// SIMATIC S7-200 project (STEP 7-Micro/WIN), CPU 224XP REL 02.01

SYMBOL_TABLE USUARIO1
PULSADOR_SUMA    I0.0     // ASCENDENTE
PULSADOR_RESTA   I0.1     // DESCENDENTE
RESET            I0.2     // RESET(REPRESENTA 0)
DISPLAY_1        MB10
DISPLAY_2        MB11
CONTADOR_1       MW2
CONTADOR_2       MW4
SEGMENTO_0_D1    Q0.0
SEGMENTO_1_D1    Q0.1
SEGMENTO_2_D1    Q0.2
SEGMENTO_3_D1    Q0.3
SEGMENTO_4_D1    Q0.4
SEGMENTO_5_D1    Q0.5
SEGMENTO_6_D1    Q0.6
SEGMENTO_0_D2    Q1.0
SEGMENTO_1_D2    Q1.1
SEGMENTO_2_D2    Q1.2
SEGMENTO_3_D2    Q1.3
SEGMENTO_4_D2    Q1.4
SEGMENTO_5_D2    Q1.5
SEGMENTO_6_D2    Q1.6
END_SYMBOL_TABLE

SYMBOL_TABLE Símbolos S7-200
Siempre_ON       SM0.0    // Siempre ON
Primer_ciclo_ON  SM0.1    // ON sólo en el primer ciclo
END_SYMBOL_TABLE

ORGANIZATION_BLOCK PRINCIPAL:OB1
TITLE=COMENTARIOS DEL PROGRAMA
BEGIN
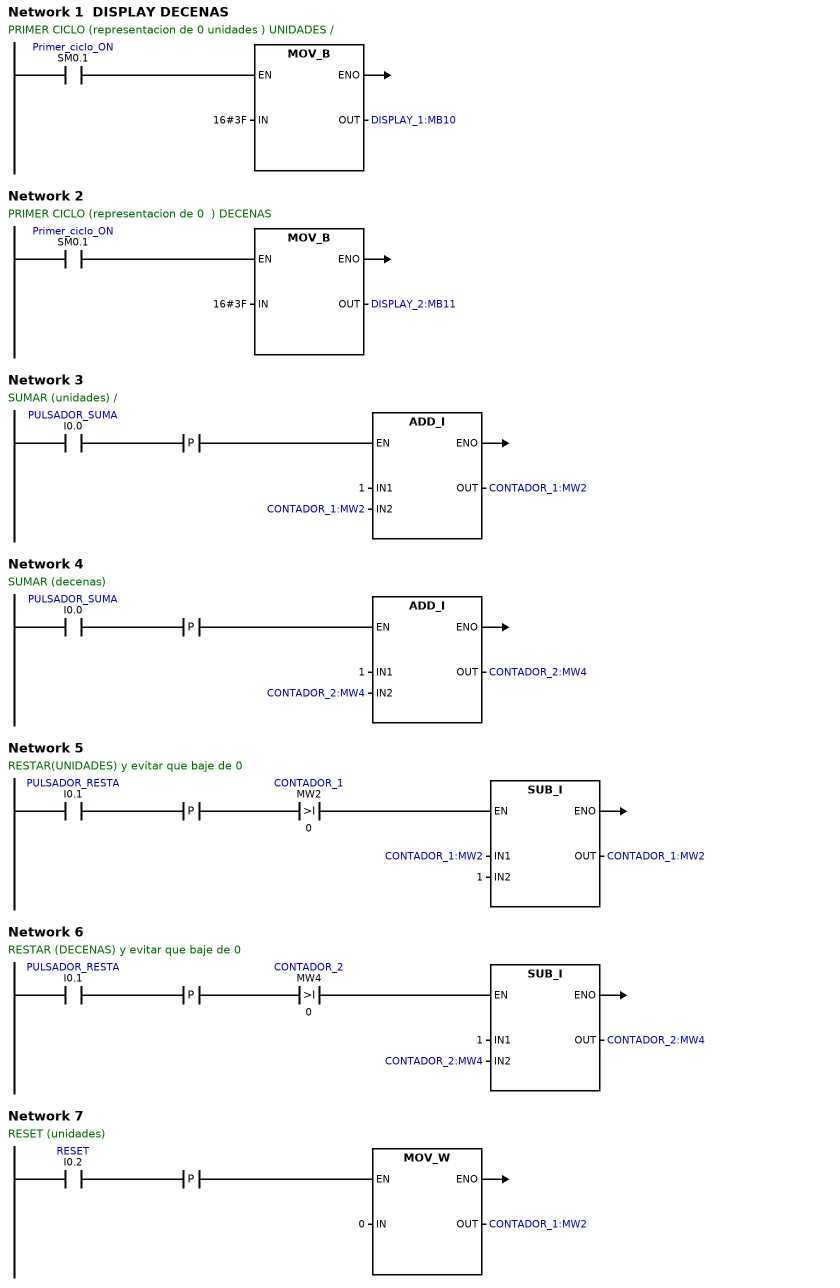
Network 1 // DISPLAY DECENAS
// PRIMER CICLO (representacion de 0 unidades ) UNIDADES
// 
LD     Primer_ciclo_ON:SM0.1
MOVB   16#3F, DISPLAY_1:MB10
Network 2
// PRIMER CICLO (representacion de 0  ) DECENAS
LD     Primer_ciclo_ON:SM0.1
MOVB   16#3F, DISPLAY_2:MB11
Network 3
// SUMAR (unidades)
// 
// (network saved uncompiled; LAD cells follow)
// row 0: c0 -| |- PULSADOR_SUMA:I0.0  c1 -|P|-  c2 --  c3 [ADD_I EN:=power@row0, IN1:=1, IN2:=CONTADOR_1:MW2, ENO=>power, OUT=>CONTADOR_1:MW2]  c4 ->
// row 1: c3 [box]
Network 4
// SUMAR (decenas)
// (network saved uncompiled; LAD cells follow)
// row 0: c0 -| |- PULSADOR_SUMA:I0.0  c1 -|P|-  c2 --  c3 [ADD_I EN:=power@row0, IN1:=1, IN2:=CONTADOR_2:MW4, ENO=>power, OUT=>CONTADOR_2:MW4]  c4 ->
// row 1: c3 [box]
Network 5
// RESTAR(UNIDADES) y evitar que baje de 0
// (network saved uncompiled; LAD cells follow)
// row 0: c0 -| |- PULSADOR_RESTA:I0.1  c1 -|P|-  c2 -|>I|- CONTADOR_1:MW2, 0  c3 --  c4 [SUB_I EN:=power@row0, IN1:=CONTADOR_1:MW2, IN2:=1, ENO=>power, OUT=>CONTADOR_1:MW2]  c5 ->
// row 1: c4 [box]
Network 6
// RESTAR (DECENAS) y evitar que baje de 0
// (network saved uncompiled; LAD cells follow)
// row 0: c0 -| |- PULSADOR_RESTA:I0.1  c1 -|P|-  c2 -|>I|- CONTADOR_2:MW4, 0  c3 --  c4 [SUB_I EN:=power@row0, IN1:=1, IN2:=CONTADOR_2:MW4, ENO=>power, OUT=>CONTADOR_2:MW4]  c5 ->
// row 1: c4 [box]
Network 7
// RESET (unidades)
// (network saved uncompiled; LAD cells follow)
// row 0: c0 -| |- RESET:I0.2  c1 -|P|-  c2 --  c3 [MOV_W EN:=power@row0, IN:=0, ENO=>power, OUT=>CONTADOR_1:MW2]  c4 ->
// row 1: c3 [box]
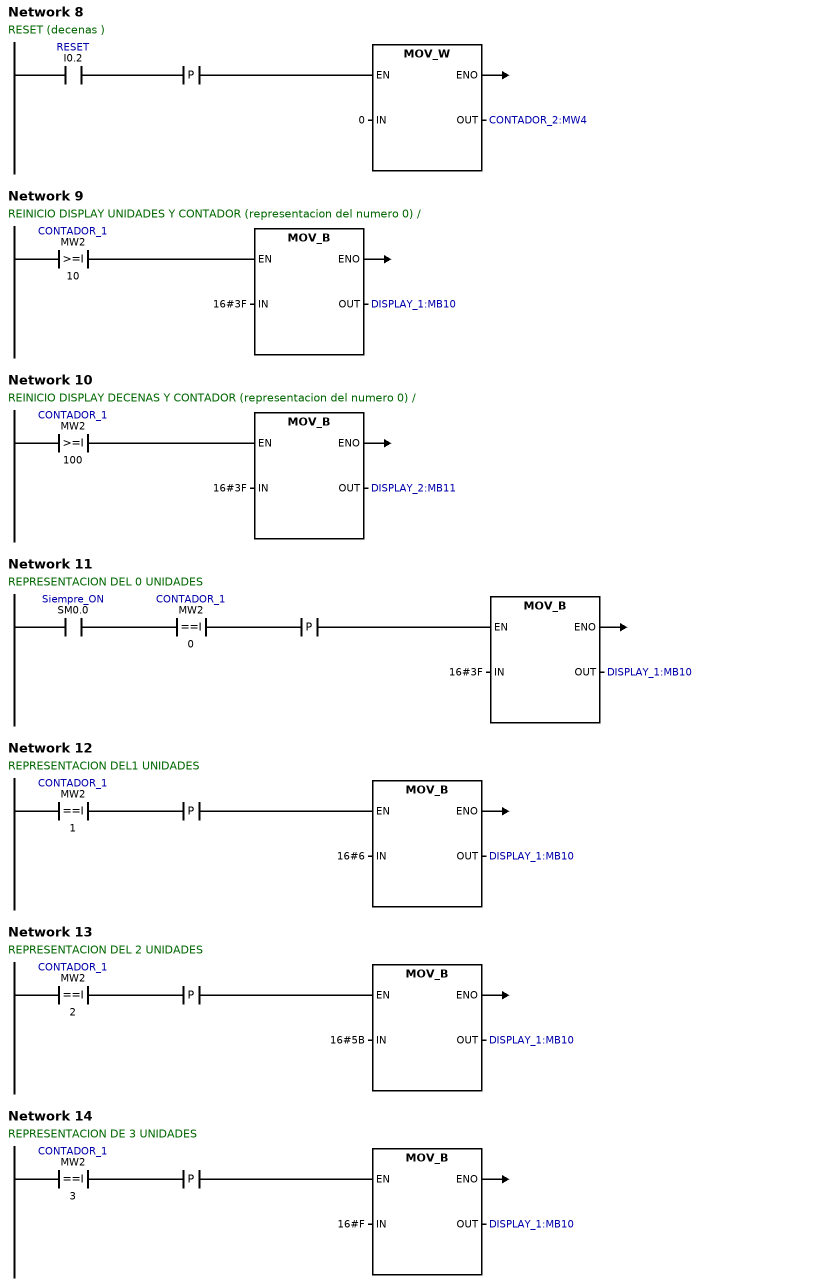
Network 8
// RESET (decenas )
// (network saved uncompiled; LAD cells follow)
// row 0: c0 -| |- RESET:I0.2  c1 -|P|-  c2 --  c3 [MOV_W EN:=power@row0, IN:=0, ENO=>power, OUT=>CONTADOR_2:MW4]  c4 ->
// row 1: c3 [box]
Network 9
// REINICIO DISPLAY UNIDADES Y CONTADOR (representacion del numero 0)
// 
// (network saved uncompiled; LAD cells follow)
// row 0: c0 -|>=I|- CONTADOR_1:MW2, 10  c1 --  c2 [MOV_B EN:=power@row0, IN:=16#3F, ENO=>power, OUT=>DISPLAY_1:MB10]  c3 ->
// row 1: c2 [box]
Network 10
// REINICIO DISPLAY DECENAS Y CONTADOR (representacion del numero 0)
// 
// (network saved uncompiled; LAD cells follow)
// row 0: c0 -|>=I|- CONTADOR_1:MW2, 100  c1 --  c2 [MOV_B EN:=power@row0, IN:=16#3F, ENO=>power, OUT=>DISPLAY_2:MB11]  c3 ->
// row 1: c2 [box]
Network 11
// REPRESENTACION DEL 0 UNIDADES
// (network saved uncompiled; LAD cells follow)
// row 0: c0 -| |- Siempre_ON:SM0.0  c1 -|==I|- CONTADOR_1:MW2, 0  c2 -|P|-  c3 --  c4 [MOV_B EN:=power@row0, IN:=16#3F, ENO=>power, OUT=>DISPLAY_1:MB10]  c5 ->
// row 1: c4 [box]
Network 12
// REPRESENTACION DEL1 UNIDADES
// (network saved uncompiled; LAD cells follow)
// row 0: c0 -|==I|- CONTADOR_1:MW2, 1  c1 -|P|-  c2 --  c3 [MOV_B EN:=power@row0, IN:=16#6, ENO=>power, OUT=>DISPLAY_1:MB10]  c4 ->
// row 1: c3 [box]
Network 13
// REPRESENTACION DEL 2 UNIDADES
// (network saved uncompiled; LAD cells follow)
// row 0: c0 -|==I|- CONTADOR_1:MW2, 2  c1 -|P|-  c2 --  c3 [MOV_B EN:=power@row0, IN:=16#5B, ENO=>power, OUT=>DISPLAY_1:MB10]  c4 ->
// row 1: c3 [box]
Network 14
// REPRESENTACION DE 3 UNIDADES
// (network saved uncompiled; LAD cells follow)
// row 0: c0 -|==I|- CONTADOR_1:MW2, 3  c1 -|P|-  c2 --  c3 [MOV_B EN:=power@row0, IN:=16#F, ENO=>power, OUT=>DISPLAY_1:MB10]  c4 ->
// row 1: c3 [box]
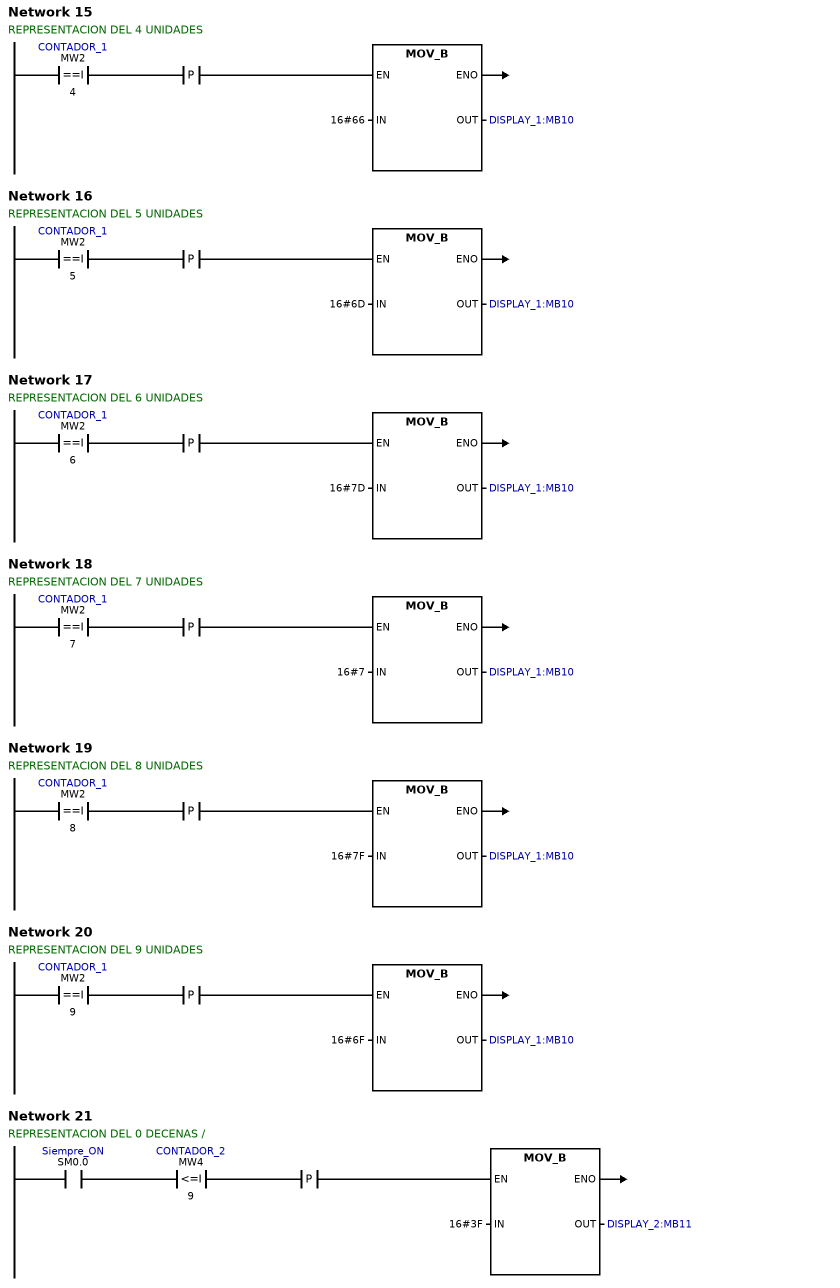
Network 15
// REPRESENTACION DEL 4 UNIDADES
// (network saved uncompiled; LAD cells follow)
// row 0: c0 -|==I|- CONTADOR_1:MW2, 4  c1 -|P|-  c2 --  c3 [MOV_B EN:=power@row0, IN:=16#66, ENO=>power, OUT=>DISPLAY_1:MB10]  c4 ->
// row 1: c3 [box]
Network 16
// REPRESENTACION DEL 5 UNIDADES
// (network saved uncompiled; LAD cells follow)
// row 0: c0 -|==I|- CONTADOR_1:MW2, 5  c1 -|P|-  c2 --  c3 [MOV_B EN:=power@row0, IN:=16#6D, ENO=>power, OUT=>DISPLAY_1:MB10]  c4 ->
// row 1: c3 [box]
Network 17
// REPRESENTACION DEL 6 UNIDADES
// (network saved uncompiled; LAD cells follow)
// row 0: c0 -|==I|- CONTADOR_1:MW2, 6  c1 -|P|-  c2 --  c3 [MOV_B EN:=power@row0, IN:=16#7D, ENO=>power, OUT=>DISPLAY_1:MB10]  c4 ->
// row 1: c3 [box]
Network 18
// REPRESENTACION DEL 7 UNIDADES
// (network saved uncompiled; LAD cells follow)
// row 0: c0 -|==I|- CONTADOR_1:MW2, 7  c1 -|P|-  c2 --  c3 [MOV_B EN:=power@row0, IN:=16#7, ENO=>power, OUT=>DISPLAY_1:MB10]  c4 ->
// row 1: c3 [box]
Network 19
// REPRESENTACION DEL 8 UNIDADES
// (network saved uncompiled; LAD cells follow)
// row 0: c0 -|==I|- CONTADOR_1:MW2, 8  c1 -|P|-  c2 --  c3 [MOV_B EN:=power@row0, IN:=16#7F, ENO=>power, OUT=>DISPLAY_1:MB10]  c4 ->
// row 1: c3 [box]
Network 20
// REPRESENTACION DEL 9 UNIDADES
// (network saved uncompiled; LAD cells follow)
// row 0: c0 -|==I|- CONTADOR_1:MW2, 9  c1 -|P|-  c2 --  c3 [MOV_B EN:=power@row0, IN:=16#6F, ENO=>power, OUT=>DISPLAY_1:MB10]  c4 ->
// row 1: c3 [box]
Network 21
// REPRESENTACION DEL 0 DECENAS
// 
// (network saved uncompiled; LAD cells follow)
// row 0: c0 -| |- Siempre_ON:SM0.0  c1 -|<=I|- CONTADOR_2:MW4, 9  c2 -|P|-  c3 --  c4 [MOV_B EN:=power@row0, IN:=16#3F, ENO=>power, OUT=>DISPLAY_2:MB11]  c5 ->
// row 1: c4 [box]
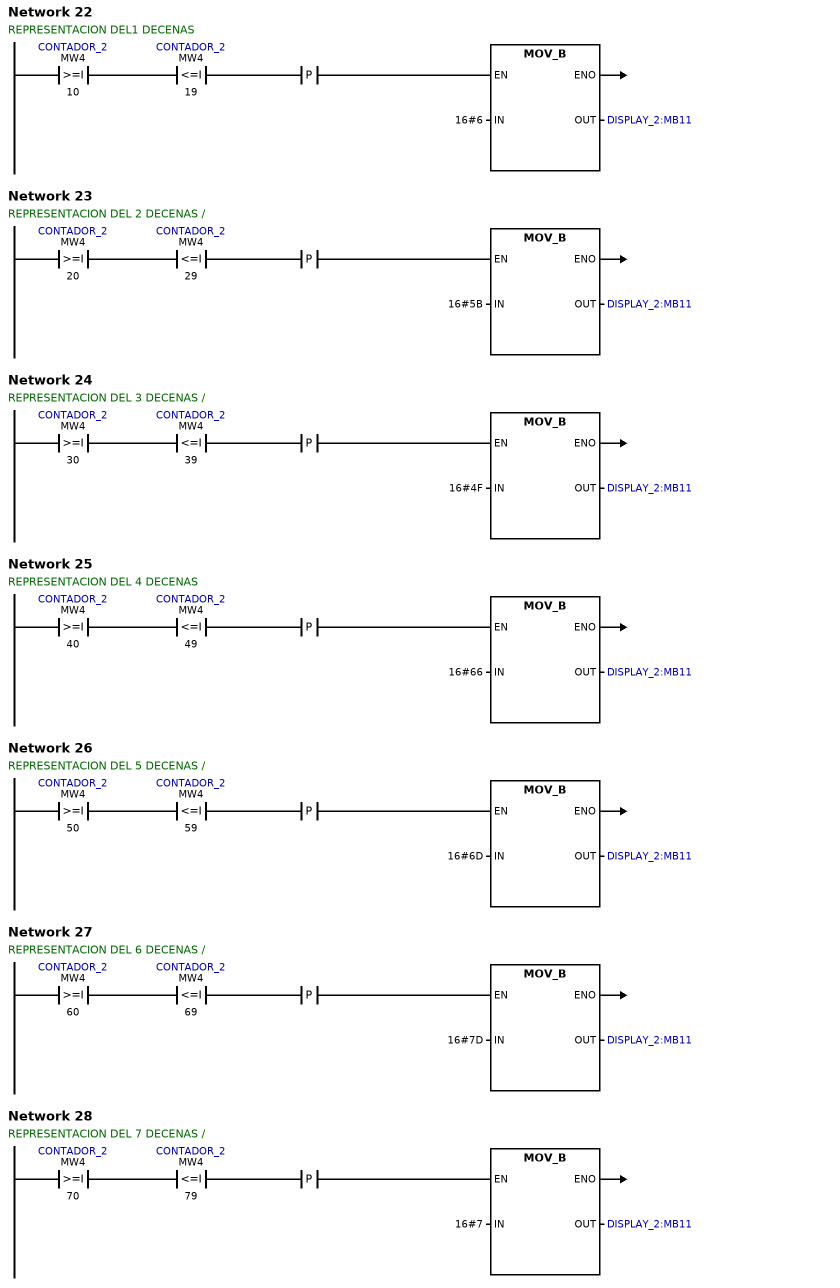
Network 22
// REPRESENTACION DEL1 DECENAS
// (network saved uncompiled; LAD cells follow)
// row 0: c0 -|>=I|- CONTADOR_2:MW4, 10  c1 -|<=I|- CONTADOR_2:MW4, 19  c2 -|P|-  c3 --  c4 [MOV_B EN:=power@row0, IN:=16#6, ENO=>power, OUT=>DISPLAY_2:MB11]  c5 ->
// row 1: c4 [box]
Network 23
// REPRESENTACION DEL 2 DECENAS
// 
// (network saved uncompiled; LAD cells follow)
// row 0: c0 -|>=I|- CONTADOR_2:MW4, 20  c1 -|<=I|- CONTADOR_2:MW4, 29  c2 -|P|-  c3 --  c4 [MOV_B EN:=power@row0, IN:=16#5B, ENO=>power, OUT=>DISPLAY_2:MB11]  c5 ->
// row 1: c4 [box]
Network 24
// REPRESENTACION DEL 3 DECENAS
// 
// (network saved uncompiled; LAD cells follow)
// row 0: c0 -|>=I|- CONTADOR_2:MW4, 30  c1 -|<=I|- CONTADOR_2:MW4, 39  c2 -|P|-  c3 --  c4 [MOV_B EN:=power@row0, IN:=16#4F, ENO=>power, OUT=>DISPLAY_2:MB11]  c5 ->
// row 1: c4 [box]
Network 25
// REPRESENTACION DEL 4 DECENAS
// (network saved uncompiled; LAD cells follow)
// row 0: c0 -|>=I|- CONTADOR_2:MW4, 40  c1 -|<=I|- CONTADOR_2:MW4, 49  c2 -|P|-  c3 --  c4 [MOV_B EN:=power@row0, IN:=16#66, ENO=>power, OUT=>DISPLAY_2:MB11]  c5 ->
// row 1: c4 [box]
Network 26
// REPRESENTACION DEL 5 DECENAS
// 
// (network saved uncompiled; LAD cells follow)
// row 0: c0 -|>=I|- CONTADOR_2:MW4, 50  c1 -|<=I|- CONTADOR_2:MW4, 59  c2 -|P|-  c3 --  c4 [MOV_B EN:=power@row0, IN:=16#6D, ENO=>power, OUT=>DISPLAY_2:MB11]  c5 ->
// row 1: c4 [box]
Network 27
// REPRESENTACION DEL 6 DECENAS
// 
// (network saved uncompiled; LAD cells follow)
// row 0: c0 -|>=I|- CONTADOR_2:MW4, 60  c1 -|<=I|- CONTADOR_2:MW4, 69  c2 -|P|-  c3 --  c4 [MOV_B EN:=power@row0, IN:=16#7D, ENO=>power, OUT=>DISPLAY_2:MB11]  c5 ->
// row 1: c4 [box]
Network 28
// REPRESENTACION DEL 7 DECENAS
// 
// (network saved uncompiled; LAD cells follow)
// row 0: c0 -|>=I|- CONTADOR_2:MW4, 70  c1 -|<=I|- CONTADOR_2:MW4, 79  c2 -|P|-  c3 --  c4 [MOV_B EN:=power@row0, IN:=16#7, ENO=>power, OUT=>DISPLAY_2:MB11]  c5 ->
// row 1: c4 [box]
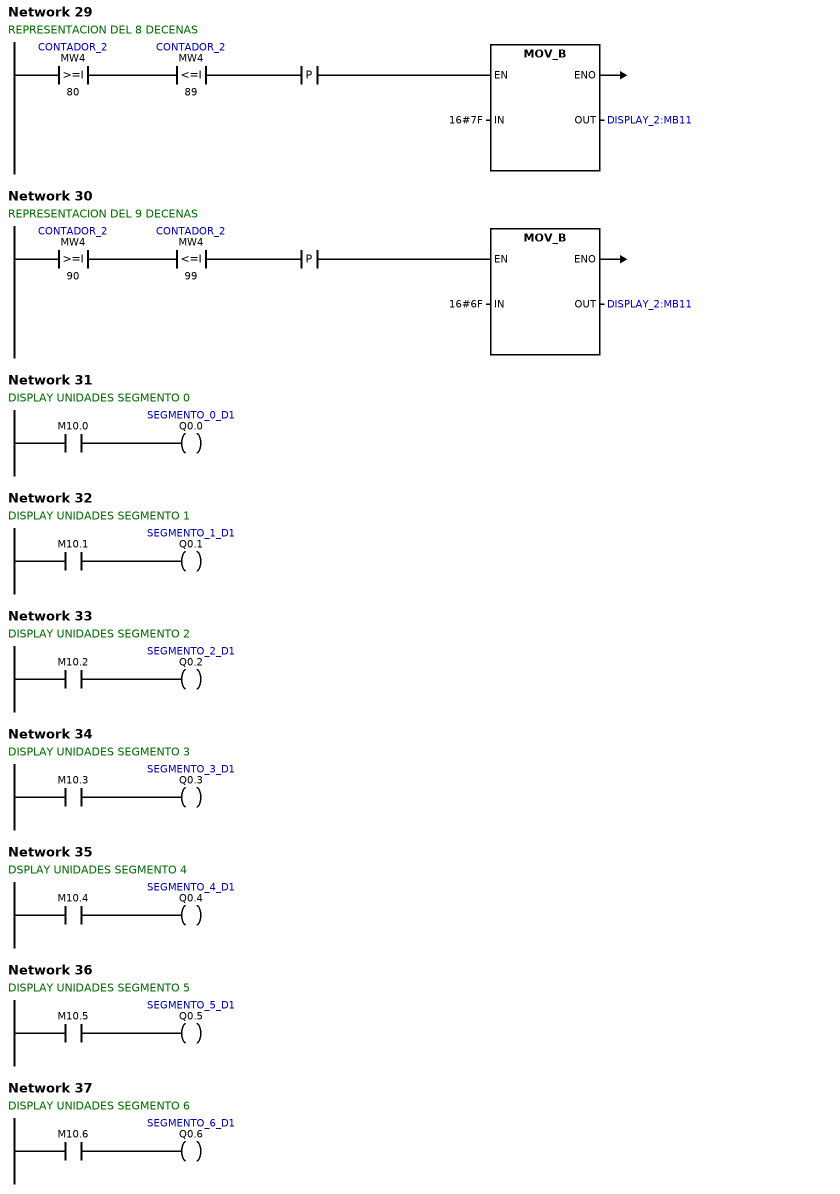
Network 29
// REPRESENTACION DEL 8 DECENAS
// (network saved uncompiled; LAD cells follow)
// row 0: c0 -|>=I|- CONTADOR_2:MW4, 80  c1 -|<=I|- CONTADOR_2:MW4, 89  c2 -|P|-  c3 --  c4 [MOV_B EN:=power@row0, IN:=16#7F, ENO=>power, OUT=>DISPLAY_2:MB11]  c5 ->
// row 1: c4 [box]
Network 30
// REPRESENTACION DEL 9 DECENAS
// (network saved uncompiled; LAD cells follow)
// row 0: c0 -|>=I|- CONTADOR_2:MW4, 90  c1 -|<=I|- CONTADOR_2:MW4, 99  c2 -|P|-  c3 --  c4 [MOV_B EN:=power@row0, IN:=16#6F, ENO=>power, OUT=>DISPLAY_2:MB11]  c5 ->
// row 1: c4 [box]
Network 31
// DISPLAY UNIDADES SEGMENTO 0
LD     M10.0
=      SEGMENTO_0_D1:Q0.0
Network 32
// DISPLAY UNIDADES SEGMENTO 1
LD     M10.1
=      SEGMENTO_1_D1:Q0.1
Network 33
// DISPLAY UNIDADES SEGMENTO 2
LD     M10.2
=      SEGMENTO_2_D1:Q0.2
Network 34
// DISPLAY UNIDADES SEGMENTO 3
LD     M10.3
=      SEGMENTO_3_D1:Q0.3
Network 35
// DSPLAY UNIDADES SEGMENTO 4
LD     M10.4
=      SEGMENTO_4_D1:Q0.4
Network 36
// DISPLAY UNIDADES SEGMENTO 5
LD     M10.5
=      SEGMENTO_5_D1:Q0.5
Network 37
// DISPLAY UNIDADES SEGMENTO 6
LD     M10.6
=      SEGMENTO_6_D1:Q0.6
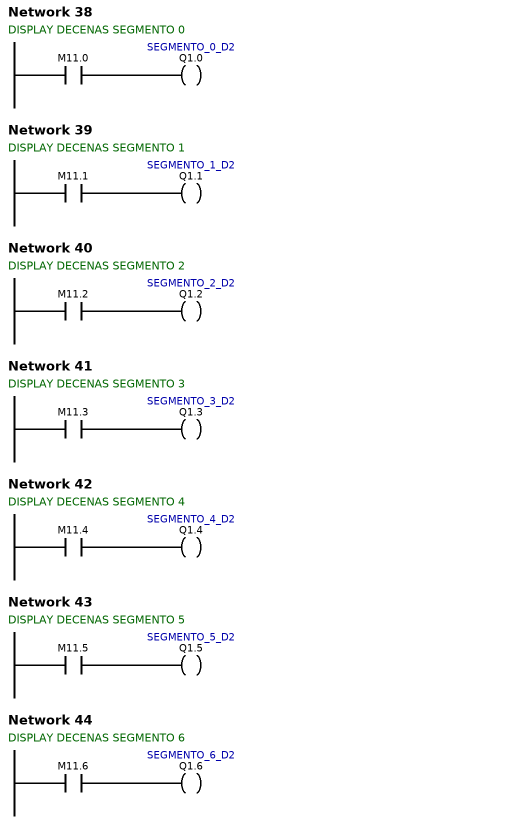
Network 38
// DISPLAY DECENAS SEGMENTO 0
LD     M11.0
=      SEGMENTO_0_D2:Q1.0
Network 39
// DISPLAY DECENAS SEGMENTO 1
LD     M11.1
=      SEGMENTO_1_D2:Q1.1
Network 40
// DISPLAY DECENAS SEGMENTO 2
LD     M11.2
=      SEGMENTO_2_D2:Q1.2
Network 41
// DISPLAY DECENAS SEGMENTO 3
LD     M11.3
=      SEGMENTO_3_D2:Q1.3
Network 42
// DISPLAY DECENAS SEGMENTO 4
LD     M11.4
=      SEGMENTO_4_D2:Q1.4
Network 43
// DISPLAY DECENAS SEGMENTO 5
LD     M11.5
=      SEGMENTO_5_D2:Q1.5
Network 44
// DISPLAY DECENAS SEGMENTO 6
LD     M11.6
=      SEGMENTO_6_D2:Q1.6
END_ORGANIZATION_BLOCK
